KUKA KRL program: ab_com_01_st01_g01_OT.src, ab_com_01_st01_g01_OT.dat

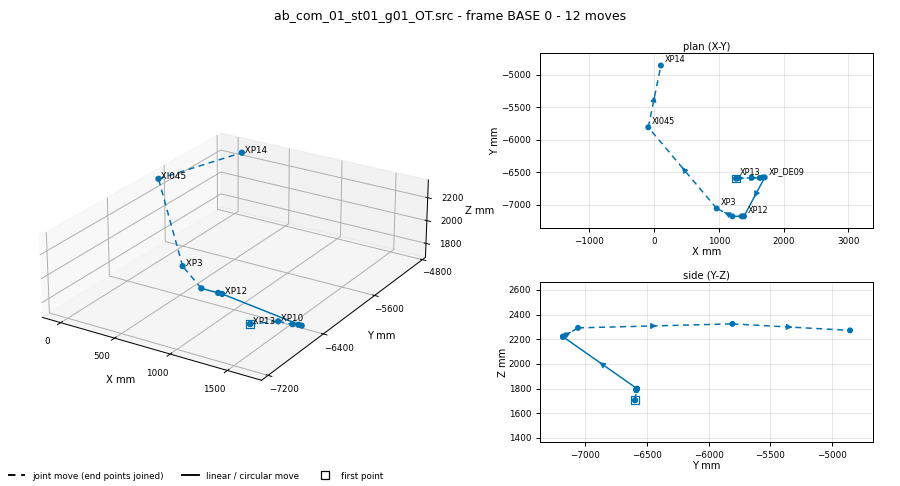
[picture p0: tool path of ab_com_01_st01_g01_OT.src in frame BASE 0, 12 of 12 moves have a stored position in this frame; points joined in program order, loops and branches not executed]
--- ab_com_01_st01_g01_OT.src ---
&ACCESS RVO1
&REL 6
&COMMENT Dep travessa LCA
&PARAM DISKPATH = KRC:\R1\Program\olp
&PARAM TEMPLATE = C:\KRC\Roboter\Template\vorgabe
&PARAM EDITMASK = *
DEF ab_com_01_st01_g01_OT( )
;FOLD INI
  ;FOLD BASISTECH INI
    GLOBAL INTERRUPT DECL 3 WHEN $STOPMESS==TRUE DO IR_STOPM ( )
    INTERRUPT ON 3
    BAS (#INITMOV,0)
  ;ENDFOLD (BASISTECH INI)
;FOLD GRIPPERTECH INI
USER_GRP(0,DUMMY,DUMMY,GDEFAULT)
;ENDFOLD (GRIPPERTECH INI)
  ;FOLD USER INI
    ;Make your modifications here

  ;ENDFOLD (USER INI)
;ENDFOLD (INI)

; Caracterizacao dos meios de producao
; Changes: Deposita LCA na GeoBox
; Modelos: Axor/Atego - ETB/LTA/LTB/STB
; Versao Atual: 30/03/2016
; Name: P13.050-R3

chk_w6_wechs_ok ( )     ; CHECK GRIPPER AXOR/ATEGO

;FOLD PTP P13 CONT Vel=100 % PDAT11 Tool[8]:Tool Changer Base[0];%{PE}%R 8.2.20,%MKUKATPBASIS,%CMOVE,%VPTP,%P 1:PTP, 2:P13, 3:C_DIS, 5:100, 7:PDAT11
$BWDSTART=FALSE
PDAT_ACT=PPDAT11
FDAT_ACT=FP13
BAS(#PTP_PARAMS,100)
PTP XP13 C_DIS
;ENDFOLD

; ABRE GRAMPOS e VERIFICA
;FOLD SET Z2.1 RPS AXOR State=OPN CONT at START Delay=1 ms;%{PE}%R 8.2.1,%MKUKATPGRP,%CGRP,%VGRP,%P 2:10, 4:1, 5:#YES, 6:GDAT26, 8:0, 10:1
TRIGGER WHEN DISTANCE=0 DELAY=1 DO H50(GRP_APO,10,1,GCONT) PRIO=-1
;ENDFOLD
;FOLD SET Z3.1 GRP AXOR State=OPN CONT at START Delay=1 ms;%{PE}%R 8.2.1,%MKUKATPGRP,%CGRP,%VGRP,%P 2:11, 4:1, 5:#YES, 6:GDAT27, 8:0, 10:1
TRIGGER WHEN DISTANCE=0 DELAY=1 DO H50(GRP_APO,11,1,GCONT) PRIO=-1
;ENDFOLD
;FOLD SET Z5.1/2/3/4 GRP AXOR State=OPN CONT at START Delay=1 ms;%{PE}%R 8.2.1,%MKUKATPGRP,%CGRP,%VGRP,%P 2:13, 4:1, 5:#YES, 6:GDAT28, 8:0, 10:1
TRIGGER WHEN DISTANCE=0 DELAY=1 DO H50(GRP_APO,13,1,GCONT) PRIO=-1
;ENDFOLD
;FOLD SET Z6.1/2/3/4 GRP AXOR State=OPN CONT at START Delay=1 ms;%{PE}%R 8.2.1,%MKUKATPGRP,%CGRP,%VGRP,%P 2:14, 4:1, 5:#YES, 6:GDAT29, 8:0, 10:1
TRIGGER WHEN DISTANCE=0 DELAY=1 DO H50(GRP_APO,14,1,GCONT) PRIO=-1
;ENDFOLD
;FOLD SET Z7.1/2 GRP AXOR State=OPN CONT at START Delay=1 ms;%{PE}%R 8.2.1,%MKUKATPGRP,%CGRP,%VGRP,%P 2:15, 4:1, 5:#YES, 6:GDAT30, 8:0, 10:1
TRIGGER WHEN DISTANCE=0 DELAY=1 DO H50(GRP_APO,15,1,GCONT) PRIO=-1
;ENDFOLD
chk_w6_rps2_opn()
chk_w6_grp3_opn()
chk_w6_grp5_opn()
chk_w6_grp6_opn()
chk_w6_grp7_opn()

;FOLD OUT 3374 'Lib. Dep. Axor/Atego' State=TRUE ;%{PE}%R 8.2.20,%MKUKATPBASIS,%COUT,%VOUTX,%P 2:3374, 3:Lib. Dep. Axor/Atego, 5:TRUE, 6:
$OUT[3374]=TRUE
;ENDFOLD
;FOLD WAIT FOR ( IN 3374 'Lib. Deposito Axor/Atego' );%{PE}%R 8.2.20,%MKUKATPBASIS,%CEXT_WAIT_FOR,%VEXT_WAIT_FOR,%P 2:, 4:, 5:$IN, 6:3374, 7:Lib. Deposito Axor/Atego, 9:
WAIT FOR  ( $IN[3374] )
;ENDFOLD
;FOLD OUT 3374 'Lib. Dep. Axor/Atego' State=FALSE ;%{PE}%R 8.2.20,%MKUKATPBASIS,%COUT,%VOUTX,%P 2:3374, 3:Lib. Dep. Axor/Atego, 5:FALSE, 6:
$OUT[3374]=FALSE
;ENDFOLD

;FOLD ; LIGA INTERLOCK 5 COM R5 com a garra rolete;%{PE}%R 8.2.20,%MKUKATPBASIS,%CCOMMENT,%VNORMAL,%P 2:LIGA  INTERLOCK  5  COM  R5  com  a  garra  rolete
;ENDFOLD
;FOLD Collision.Monitoring_5_On ;%{PE}%MKUKATPUSER
COLLSTOP( 5, 1 ) ;Interrupt-Controlled
;ENDFOLD

;FOLD PTP P9 CONT Vel=100 % PDAT7 Tool[8]:Tool Changer Base[0];%{PE}%R 8.2.20,%MKUKATPBASIS,%CMOVE,%VPTP,%P 1:PTP, 2:P9, 3:C_DIS, 5:100, 7:PDAT7
$BWDSTART=FALSE
PDAT_ACT=PPDAT7
FDAT_ACT=FP9
BAS(#PTP_PARAMS,100)
PTP XP9 C_DIS
;ENDFOLD
;FOLD PTP P10 CONT Vel=100 % PDAT8 Tool[8]:Tool Changer Base[0];%{PE}%R 8.2.20,%MKUKATPBASIS,%CMOVE,%VPTP,%P 1:PTP, 2:P10, 3:C_DIS, 5:100, 7:PDAT8
$BWDSTART=FALSE
PDAT_ACT=PPDAT8
FDAT_ACT=FP10
BAS(#PTP_PARAMS,100)
PTP XP10 C_DIS
;ENDFOLD

; VERIFICA PRESENCA LCA OK
IF (NOT(GHOST())) THEN
;FOLD WAIT FOR ( IN 489 'Presença de peça 1 - Axor LCA' );%{PE}%R 8.2.20,%MKUKATPBASIS,%CEXT_WAIT_FOR,%VEXT_WAIT_FOR,%P 2:, 4:, 5:$IN, 6:489, 7:Presença de peça 1 - Axor LCA, 9:
WAIT FOR  ( $IN[489] )
;ENDFOLD
ENDIF

; ABRE GRAMPO Z4.1 "LCA"
;FOLD SET Z4.1 GRP AXOR State=OPN CONT at START Delay=1 ms;%{PE}%R 8.2.1,%MKUKATPGRP,%CGRP,%VGRP,%P 2:12, 4:1, 5:#YES, 6:GDAT32, 8:0, 10:1
TRIGGER WHEN DISTANCE=0 DELAY=1 DO H50(GRP_APO,12,1,GCONT) PRIO=-1
;ENDFOLD

;FOLD PTP l035 CONT Vel=100 % P_OLP8 Tool[8]:Tool Changer Base[0];%{PE}%R 8.2.20,%MKUKATPBASIS,%CMOVE,%VPTP,%P 1:PTP, 2:l035, 3:C_DIS, 5:100, 7:P_OLP8
$BWDSTART=FALSE
PDAT_ACT=PP_OLP8
FDAT_ACT=Fl035
BAS(#PTP_PARAMS,100)
PTP Xl035 C_DIS
;ENDFOLD
;FOLD LIN P1 CONT Vel=0.5 m/s CPDAT1 Tool[8]:Tool Changer Base[0];%{PE}%R 8.2.20,%MKUKATPBASIS,%CMOVE,%VLIN,%P 1:LIN, 2:P1, 3:C_DIS C_DIS, 5:0.5, 7:CPDAT1
$BWDSTART=FALSE
LDAT_ACT=LCPDAT1
FDAT_ACT=FP1
BAS(#CP_PARAMS,0.5)
LIN XP1 C_DIS C_DIS
;ENDFOLD

; VERIFICA GRAMPO Z4.1 ABERTO
chk_w6_grp4_opn( )

;FOLD ; Posicao de deposito Gripper AXOR;%{PE}%R 8.2.20,%MKUKATPBASIS,%CCOMMENT,%VNORMAL,%P 2:Posicao de deposito Gripper AXOR
;ENDFOLD
;FOLD LIN P_DE09  Vel=0.25 m/s L_OLP1 Tool[6]:Gripper AXOR Base[0];%{PE}%R8.2.19,%MKUKATPBASIS,%CMOVE,%VLIN,%P 1:LIN, 2:P_DE09, 3: , 5:0.25, 7:L_OLP1
$BWDSTART = FALSE
LDAT_ACT= LL_OLP1
FDAT_ACT= FP_DE09
BAS(#CP_PARAMS,0.25)
LIN XP_DE09
;ENDFOLD

IF (NOT(GHOST())) THEN
;FOLD WAIT FOR ( IN 490 'Presença de peça 2 - Axor' AND IN 491 'Presença de peça 3 - Axor' AND IN 492 'Presença de peça 4 - Axor' );%{PE}%R 8.2.20,%MKUKATPBASIS,%CEXT_WAIT_FOR,%VEXT_WAIT_FOR,%P 2:, 4:, 5:$IN, 6:490, 7:Presença de peça 2 - Axor, 8:AND, 9:, 10:$IN, 11:491, 12:Presença de peça 3 - Axor, 13:AND, 14:, 15:$IN, 16:492, 17:Presença de peça 4 - Axor, 19:
WAIT FOR  ( $IN[490] AND $IN[491] AND $IN[492] )
;ENDFOLD
ENDIF

;FOLD OUT 3375 'Lib. p/ sair s/ Gripper Axor/Atego' State=TRUE ;%{PE}%R 8.2.20,%MKUKATPBASIS,%COUT,%VOUTX,%P 2:3375, 3:Lib. p/ sair s/ Gripper Axor/Atego, 5:TRUE, 6:
$OUT[3375]=TRUE
;ENDFOLD

; VERIFICA PRESENCA LCA OK
IF (NOT(GHOST())) THEN
;FOLD WAIT FOR ( IN 489 'Presença de peça 1 - Axor LCA' );%{PE}%R 8.2.20,%MKUKATPBASIS,%CEXT_WAIT_FOR,%VEXT_WAIT_FOR,%P 2:, 4:, 5:$IN, 6:489, 7:Presença de peça 1 - Axor LCA, 9:
WAIT FOR  ( $IN[489] )
;ENDFOLD
ENDIF

; FECHA GRAMPOS
;FOLD SET Z2.1 RPS AXOR State=CLO GDAT15;%{PE}%R 8.2.1,%MKUKATPGRP,%CGRP,%VGRP,%P 2:10, 4:2, 5:#NO, 6:GDAT15, 8:0, 10:0
H50(GRP,10,2,GGDAT15)
;ENDFOLD
;FOLD SET Z3.1 GRP AXOR State=CLO GDAT8;%{PE}%R 8.2.1,%MKUKATPGRP,%CGRP,%VGRP,%P 2:11, 4:2, 5:#NO, 6:GDAT8, 8:0, 10:0
H50(GRP,11,2,GGDAT8)
;ENDFOLD
;FOLD SET Z5.1/2/3/4 GRP AXOR State=CLO GDAT16;%{PE}%R 8.2.1,%MKUKATPGRP,%CGRP,%VGRP,%P 2:13, 4:2, 5:#NO, 6:GDAT16, 8:0, 10:0
H50(GRP,13,2,GGDAT16)
;ENDFOLD
;FOLD SET Z6.1/2/3/4 GRP AXOR State=CLO GDAT17;%{PE}%R 8.2.1,%MKUKATPGRP,%CGRP,%VGRP,%P 2:14, 4:2, 5:#NO, 6:GDAT17, 8:0, 10:0
H50(GRP,14,2,GGDAT17)
;ENDFOLD

; VERIFICA GRAMPOS FECHADOS
chk_w6_rps2_clo( )
chk_w6_grp3_clo( )

; FECHA GRAMPOS Z4.1 e Z7.1
;FOLD SET Z4.1 GRP AXOR State=CLO GDAT31;%{PE}%R 8.2.1,%MKUKATPGRP,%CGRP,%VGRP,%P 2:12, 4:2, 5:#NO, 6:GDAT31, 8:0, 10:0
H50(GRP,12,2,GGDAT31)
;ENDFOLD
;FOLD SET Z7.1/2 GRP AXOR State=CLO GDAT33;%{PE}%R 8.2.1,%MKUKATPGRP,%CGRP,%VGRP,%P 2:15, 4:2, 5:#NO, 6:GDAT33, 8:0, 10:0
H50(GRP,15,2,GGDAT33)
;ENDFOLD
;FOLD SET VACUO AXOR State=BLOW GDAT34;%{PE}%R 8.2.1,%MKUKATPGRP,%CGRP,%VGRP,%P 2:9, 4:2, 5:#NO, 6:GDAT34, 8:0, 10:0
H50(GRP,9,2,GGDAT34)
;ENDFOLD
;FOLD SET VACUO AXOR State=OFF GDAT35;%{PE}%R 8.2.1,%MKUKATPGRP,%CGRP,%VGRP,%P 2:9, 4:3, 5:#NO, 6:GDAT35, 8:0, 10:0
H50(GRP,9,3,GGDAT35)
;ENDFOLD

; VERIFICA GRAMPOS FECHADOS
chk_w6_grp5_clo( )
chk_w6_grp6_clo( )
chk_w6_grp7_clo( )
chk_w6_grp4_clo( )
chk_w6_grp1_vacoff( )

; VERIFICA PRESENCA LCA OK
IF (NOT(GHOST())) THEN
;FOLD WAIT FOR ( IN 489 'Presença de peça 1 - Axor LCA' );%{PE}%R 8.2.20,%MKUKATPBASIS,%CEXT_WAIT_FOR,%VEXT_WAIT_FOR,%P 2:, 4:, 5:$IN, 6:489, 7:Presença de peça 1 - Axor LCA, 9:
WAIT FOR  ( $IN[489] )
;ENDFOLD
ENDIF

;FOLD OUT 3375 'Lib. p/ sair s/ Gripper Axor/Atego' State=TRUE ;%{PE}%R 8.2.20,%MKUKATPBASIS,%COUT,%VOUTX,%P 2:3375, 3:Lib. p/ sair s/ Gripper Axor/Atego, 5:TRUE, 6:
$OUT[3375]=TRUE
;ENDFOLD
;FOLD WAIT FOR ( IN 3375 'Lib. p/ sair s/ Gripper Axor/Atego' );%{PE}%R 8.2.20,%MKUKATPBASIS,%CEXT_WAIT_FOR,%VEXT_WAIT_FOR,%P 2:, 4:, 5:$IN, 6:3375, 7:Lib. p/ sair s/ Gripper Axor/Atego, 9:
WAIT FOR  ( $IN[3375] )
;ENDFOLD
;FOLD OUT 3375 'Lib. p/ sair s/ Gripper Axor/Atego' State=FALSE ;%{PE}%R 8.2.20,%MKUKATPBASIS,%COUT,%VOUTX,%P 2:3375, 3:Lib. p/ sair s/ Gripper Axor/Atego, 5:FALSE, 6:
$OUT[3375]=FALSE
;ENDFOLD

;FOLD WAIT Time=0.5 sec;%{PE}%R 8.2.20,%MKUKATPBASIS,%CWAIT,%VWAIT,%P 3:0.5
WAIT SEC 0.5
;ENDFOLD
;FOLD OUT 224 'Bloquear MPS' State=FALSE ;%{PE}%R 8.2.20,%MKUKATPBASIS,%COUT,%VOUTX,%P 2:224, 3:Bloquear MPS, 5:FALSE, 6:
$OUT[224]=FALSE
;ENDFOLD
;FOLD OUT 223 'Desbloquear MPS' State=TRUE ;%{PE}%R 8.2.20,%MKUKATPBASIS,%COUT,%VOUTX,%P 2:223, 3:Desbloquear MPS, 5:TRUE, 6:
$OUT[223]=TRUE
;ENDFOLD
;FOLD WAIT FOR ( IN 217 'MPS Destravado' );%{PE}%R 8.2.20,%MKUKATPBASIS,%CEXT_WAIT_FOR,%VEXT_WAIT_FOR,%P 2:, 4:, 5:$IN, 6:217, 7:MPS Destravado, 9:
WAIT FOR  ( $IN[217] )
;ENDFOLD
;FOLD WAIT FOR NOT ( IN 221 'MPS Travado' );%{PE}%R 8.2.20,%MKUKATPBASIS,%CEXT_WAIT_FOR,%VEXT_WAIT_FOR,%P 2:NOT, 4:, 5:$IN, 6:221, 7:MPS Travado, 9:
WAIT FOR  NOT ( $IN[221] )
;ENDFOLD
;FOLD IBUS OFF;%{PE}%R 8.2.20,%MKUKATPBASIS,%CIBUS,%VMAP,%P 2:#OFF, 3:3
$IBUS_OFF=$IBUS_ON
$IBUS_ON=0
;ENDFOLD
;FOLD WAIT Time=0.5 sec;%{PE}%R 8.2.20,%MKUKATPBASIS,%CWAIT,%VWAIT,%P 3:0.5
WAIT SEC 0.5
;ENDFOLD

;FOLD LIN P12 Vel=0.25 m/s CPDAT6 Tool[8]:Tool Changer Base[0];%{PE}%R 8.2.20,%MKUKATPBASIS,%CMOVE,%VLIN,%P 1:LIN, 2:P12, 3:, 5:0.25, 7:CPDAT6
$BWDSTART=FALSE
LDAT_ACT=LCPDAT6
FDAT_ACT=FP12
BAS(#CP_PARAMS,0.25)
LIN XP12
;ENDFOLD

;FOLD WAIT FOR NOT ( IN 219 'Posicao p/ Acoplamento OK' );%{PE}%R 8.2.20,%MKUKATPBASIS,%CEXT_WAIT_FOR,%VEXT_WAIT_FOR,%P 2:NOT, 4:, 5:$IN, 6:219, 7:Posicao p/ Acoplamento OK, 9:
WAIT FOR  NOT ( $IN[219] )
;ENDFOLD

;FOLD LIN l040 Vel=0.25 m/s L_OLP2 Tool[8]:Tool Changer Base[0];%{PE}%R 8.2.20,%MKUKATPBASIS,%CMOVE,%VLIN,%P 1:LIN, 2:l040, 3:, 5:0.25, 7:L_OLP2
$BWDSTART=FALSE
LDAT_ACT=LL_OLP2
FDAT_ACT=Fl040
BAS(#CP_PARAMS,0.25)
LIN Xl040
;ENDFOLD

;FOLD WAIT FOR NOT ( IN 219 'Posicao p/ Acoplamento OK' );%{PE}%R 8.2.20,%MKUKATPBASIS,%CEXT_WAIT_FOR,%VEXT_WAIT_FOR,%P 2:NOT, 4:, 5:$IN, 6:219, 7:Posicao p/ Acoplamento OK, 9:
WAIT FOR  NOT ( $IN[219] )
;ENDFOLD
;FOLD OUT 223 'Desbloquear MPS' State=FALSE ;%{PE}%R 8.2.20,%MKUKATPBASIS,%COUT,%VOUTX,%P 2:223, 3:Desbloquear MPS, 5:FALSE, 6:
$OUT[223]=FALSE
;ENDFOLD

;FOLD LIN P2 CONT Vel=1 m/s CPDAT2 Tool[8]:Tool Changer Base[0];%{PE}%R 8.2.20,%MKUKATPBASIS,%CMOVE,%VLIN,%P 1:LIN, 2:P2, 3:C_DIS C_DIS, 5:1, 7:CPDAT2
$BWDSTART=FALSE
LDAT_ACT=LCPDAT2
FDAT_ACT=FP2
BAS(#CP_PARAMS,1)
LIN XP2 C_DIS C_DIS
;ENDFOLD
;FOLD PTP P3 CONT Vel=100 % PDAT1 Tool[8]:Tool Changer Base[0];%{PE}%R 8.2.20,%MKUKATPBASIS,%CMOVE,%VPTP,%P 1:PTP, 2:P3, 3:C_DIS, 5:100, 7:PDAT1
$BWDSTART=FALSE
PDAT_ACT=PPDAT1
FDAT_ACT=FP3
BAS(#PTP_PARAMS,100)
PTP XP3 C_DIS
;ENDFOLD
;FOLD PTP l045 CONT Vel=100 % P_OLP9 Tool[8]:Tool Changer Base[0];%{PE}%R 8.2.20,%MKUKATPBASIS,%CMOVE,%VPTP,%P 1:PTP, 2:l045, 3:C_DIS, 5:100, 7:P_OLP9
$BWDSTART=FALSE
PDAT_ACT=PP_OLP9
FDAT_ACT=Fl045
BAS(#PTP_PARAMS,100)
PTP Xl045 C_DIS
;ENDFOLD

;FOLD PULSE 3343 'R3 entregou peça Geo' State=TRUE Time=3 sec;%{PE}%R 8.2.20,%MKUKATPBASIS,%COUT,%VPULSE,%P 2:3343, 3:R3 entregou peça Geo, 5:TRUE, 6:, 8:3
PULSE($OUT[3343], TRUE,3)
;ENDFOLD

;FOLD PTP P14 CONT Vel=100 % PDAT12 Tool[8]:Tool Changer Base[0];%{PE}%R 8.2.20,%MKUKATPBASIS,%CMOVE,%VPTP,%P 1:PTP, 2:P14, 3:C_DIS, 5:100, 7:PDAT12
$BWDSTART=FALSE
PDAT_ACT=PPDAT12
FDAT_ACT=FP14
BAS(#PTP_PARAMS,100)
PTP XP14 C_DIS
;ENDFOLD

;FOLD ; DESLIGA INTERLOCK 1 COM R1 NA PEGA DA GARRA 913;%{PE}%R 8.2.20,%MKUKATPBASIS,%CCOMMENT,%VNORMAL,%P 2:DESLIGA  INTERLOCK  1  COM  R1  NA  PEGA  DA  GARRA  913
;ENDFOLD
;FOLD Collision.Monitoring_1_Off . ;%{PE}%MKUKATPUSER
COLLSTOP( 1, 2+0 )
;ENDFOLD

;FOLD ; DESLIGA INTERLOCK 5 COM R5;%{PE}%R 8.2.20,%MKUKATPBASIS,%CCOMMENT,%VNORMAL,%P 2:DESLIGA  INTERLOCK  5  COM  R5
;ENDFOLD
;FOLD Collision.Monitoring_5_Off . ;%{PE}%MKUKATPUSER
COLLSTOP( 5, 2+0 )
;ENDFOLD

;FOLD OUT 3374 'Lib. Dep. Axor/Atego' State=TRUE ;%{PE}%R 8.2.20,%MKUKATPBASIS,%COUT,%VOUTX,%P 2:3374, 3:Lib. Dep. Axor/Atego, 5:TRUE, 6:
$OUT[3374]=TRUE
;ENDFOLD
;FOLD OUT 3348 'Fora area GEOBOX' State=TRUE ;%{PE}%R 8.2.20,%MKUKATPBASIS,%COUT,%VOUTX,%P 2:3348, 3:Fora area GEOBOX, 5:TRUE, 6:
$OUT[3348]=TRUE
;ENDFOLD

END

--- ab_com_01_st01_g01_OT.dat ---
&ACCESS RVO1
&REL 6
&COMMENT Dep travessa LCA
&PARAM DISKPATH = KRC:\R1\Program\olp
&PARAM TEMPLATE = C:\KRC\Roboter\Template\vorgabe
&PARAM EDITMASK = *
DEFDAT  ab_com_01_st01_g01_OT
;FOLD EXTERNAL DECLARATIONS;%{PE}%MKUKATPBASIS,%CEXT,%VCOMMON,%P
;FOLD GRIPPERTECH EXT
EXT  H50 (INT  :IN,INT  :IN,INT  :IN,GRP_TYP  :IN )
;ENDFOLD (GRIPPERTECH EXT)
;FOLD SPOTTECH EXT

;ENDFOLD (SPOTTECH EXT)
;FOLD BASISTECH EXT;%{PE}%MKUKATPBASIS,%CEXT,%VEXT,%P
EXT  BAS (BAS_COMMAND  :IN,REAL  :IN )
DECL INT SUCCESS
;ENDFOLD (BASISTECH EXT)
;FOLD USER EXT;%{E}%MKUKATPUSER,%CEXT,%VEXT,%P
;Make your modifications here

;ENDFOLD (USER EXT)
;ENDFOLD (EXTERNAL DECLARATIONS)
DECL FDAT Fl035={TOOL_NO 6,BASE_NO 0,IPO_FRAME #BASE,POINT2[] " "}
DECL PDAT PP_OLP8={VEL 100.0,ACC 100.0,APO_DIST 100.0,APO_MODE #CDIS}
DECL E6POS Xl035={X 1631.40002,Y -6588.3291,Z 1794.03101,A 70.7797089,B -89.9868469,C -175.781799,S 6,T 51,E1 5700.0,E2 0.0,E3 0.0,E4 0.0,E5 0.0,E6 0.0}
DECL FDAT FP_DE09={TOOL_NO 6,BASE_NO 0,IPO_FRAME #BASE,POINT2[] " "}
DECL E6POS XP_DE09={X 1707.35596,Y -6580.3291,Z 1798.76196,A -108.196297,B -89.8673096,C 3.225034,S 6,T 51,E1 5699.99805,E2 0.0,E3 0.0,E4 0.0,E5 0.0,E6 0.0}
DECL LDAT LL_OLP1={VEL 0.25,ACC 100.0,APO_DIST 0.0,APO_FAC 0.0,ORI_TYP #VAR,CIRC_TYP #BASE,JERK_FAC 50.0}
DECL FDAT Fl040={TOOL_NO 8,BASE_NO 0,IPO_FRAME #BASE,POINT2[] " ",TQ_STATE FALSE}
DECL E6POS Xl040={X 1353.49902,Y -7181.71094,Z 2220.25488,A -90.1084976,B -74.8772964,C -89.8598785,S 6,T 51,E1 5700.01904,E2 0.0,E3 0.0,E4 0.0,E5 0.0,E6 0.0}
DECL LDAT LL_OLP2={VEL 0.25,ACC 100.0,APO_DIST 20.0,APO_FAC 0.0,ORI_TYP #VAR,CIRC_TYP #BASE,JERK_FAC 50.0}
DECL FDAT Fl045={TOOL_NO 8,BASE_NO 0,IPO_FRAME #BASE,POINT2[] " "}
DECL PDAT PP_OLP9={VEL 100.0,ACC 100.0,APO_DIST 100.0,APO_MODE #CDIS}
DECL E6POS Xl045={X -89.0451508,Y -5808.14014,Z 2324.49902,A 10.4492998,B 8.6899004,C 149.959503,S 6,T 51,E1 4593.48291,E2 0.0,E3 0.0,E4 0.0,E5 0.0,E6 0.0}
DECL BASIS_SUGG_T LAST_BASIS={POINT1[] "P0                      ",POINT2[] "P0                      ",CP_PARAMS[] "CPDAT0                  ",PTP_PARAMS[] "PDAT0                   ",CONT[] "                        ",CP_VEL[] "2.0                     ",PTP_VEL[] " 100                    ",SYNC_PARAMS[] "SYNCDAT                 ",SPL_NAME[] "S0                      "}
DECL E6POS XP1={X 1678.87805,Y -6580.3291,Z 1798.76196,A -108.197998,B -89.8673096,C 3.226717,S 6,T 51,E1 5699.99805,E2 0.0,E3 0.0,E4 0.0,E5 0.0,E6 0.0}
DECL FDAT FP1={TOOL_NO 6,BASE_NO 0,IPO_FRAME #BASE,POINT2[] " ",TQ_STATE FALSE}
DECL LDAT LCPDAT1={VEL 2.0,ACC 100.0,APO_DIST 50.0,APO_FAC 50.0,AXIS_VEL 100.0,AXIS_ACC 100.0,ORI_TYP #VAR,CIRC_TYP #BASE,JERK_FAC 50.0,GEAR_JERK 50.0,EXAX_IGN 0}
DECL E6POS XP2={X 1208.60706,Y -7181.56104,Z 2220.479,A -89.9195328,B -74.9438934,C -90.0642395,S 6,T 51,E1 5699.41699,E2 0.0,E3 0.0,E4 0.0,E5 0.0,E6 0.0}
DECL FDAT FP2={TOOL_NO 8,BASE_NO 0,IPO_FRAME #BASE,POINT2[] " ",TQ_STATE FALSE}
DECL LDAT LCPDAT2={VEL 2.0,ACC 100.0,APO_DIST 100.0,APO_FAC 50.0,AXIS_VEL 100.0,AXIS_ACC 100.0,ORI_TYP #VAR,CIRC_TYP #BASE,JERK_FAC 50.0,GEAR_JERK 50.0,EXAX_IGN 0}
DECL E6POS XP3={X 965.776001,Y -7059.44189,Z 2292.1189,A -54.9305382,B -71.0292969,C -129.947205,S 6,T 51,E1 5619.95313,E2 0.0,E3 0.0,E4 0.0,E5 0.0,E6 0.0}
DECL FDAT FP3={TOOL_NO 8,BASE_NO 0,IPO_FRAME #BASE,POINT2[] " ",TQ_STATE FALSE}
DECL PDAT PPDAT1={VEL 100.0,ACC 100.0,APO_DIST 100.0,APO_MODE #CDIS}
DECL GRP_SUGG_T LAST_GRP={NUMBER[] "9                       ",STATE[] "3                       ",PARAMS[] "GDAT35                  "}
DECL GRP_TYP GGDAT2={G_APO #NO,GRP_TIME 0.200000003,CTRL #OFF,DLY 0,DST 1}
DECL GRP_TYP GGDAT1={G_APO #NO,GRP_TIME 0.200000003,CTRL #OFF,DLY 0,DST 1}
DECL GRP_TYP GGDAT3={G_APO #NO,GRP_TIME 0.200000003,CTRL #OFF,DLY 0,DST 1}
DECL GRP_TYP GGDAT4={G_APO #NO,GRP_TIME 0.200000003,CTRL #OFF,DLY 0,DST 1}
DECL GRP_TYP GGDAT5={G_APO #NO,GRP_TIME 0.200000003,CTRL #OFF,DLY 0,DST 1}
DECL GRP_TYP GGDAT6={G_APO #NO,GRP_TIME 0.200000003,CTRL #OFF,DLY 0,DST 1}
DECL GRP_TYP GGDAT7={G_APO #NO,GRP_TIME 0.200000003,CTRL #OFF,DLY 0,DST 1}
DECL GRP_TYP GGDAT8={G_APO #NO,GRP_TIME 0.200000003,CTRL #OFF,DLY 0,DST 1}
DECL GRP_TYP GGDAT9={G_APO #NO,GRP_TIME 0.200000003,CTRL #OFF,DLY 0,DST 1}
DECL GRP_TYP GGDAT10={G_APO #NO,GRP_TIME 0.200000003,CTRL #OFF,DLY 0,DST 1}
DECL GRP_TYP GGDAT11={G_APO #NO,GRP_TIME 0.200000003,CTRL #OFF,DLY 0,DST 1}
DECL GRP_TYP GGDAT12={G_APO #NO,GRP_TIME 0.200000003,CTRL #OFF,DLY 0,DST 1}
DECL GRP_TYP GGDAT13={G_APO #NO,GRP_TIME 0.200000003,CTRL #OFF,DLY 0,DST 1}
DECL GRP_TYP GGDAT14={G_APO #NO,GRP_TIME 0.200000003,CTRL #OFF,DLY 0,DST 1}
DECL GRP_TYP GGDAT15={G_APO #NO,GRP_TIME 0.200000003,CTRL #OFF,DLY 0,DST 1}
DECL GRP_TYP GGDAT16={G_APO #NO,GRP_TIME 0.200000003,CTRL #OFF,DLY 0,DST 1}
DECL GRP_TYP GGDAT17={G_APO #NO,GRP_TIME 0.200000003,CTRL #OFF,DLY 0,DST 1}
DECL GRP_TYP GGDAT18={G_APO #NO,GRP_TIME 0.200000003,CTRL #OFF,DLY 0,DST 1}
DECL GRP_TYP GGDAT19={G_APO #NO,GRP_TIME 0.200000003,CTRL #OFF,DLY 0,DST 1}
DECL E6POS XP8={X 846.208923,Y -6811.92188,Z 1735.02002,A -9.90643406,B -75.1019363,C -110.246101,S 6,T 51,E1 5398.51416,E2 0.0,E3 0.0,E4 0.0,E5 0.0,E6 0.0}
DECL FDAT FP8={TOOL_NO 6,BASE_NO 0,IPO_FRAME #BASE,POINT2[] " ",TQ_STATE FALSE}
DECL PDAT PPDAT6={VEL 100.0,ACC 100.0,APO_DIST 100.0,APO_MODE #CDIS}
DECL E6POS XP9={X 1266.59302,Y -6597.0752,Z 1705.35596,A 1.41324604,B -82.7240829,C -106.323402,S 6,T 51,E1 5699.94922,E2 0.0,E3 0.0,E4 0.0,E5 0.0,E6 0.0}
DECL FDAT FP9={TOOL_NO 6,BASE_NO 0,IPO_FRAME #BASE,POINT2[] " ",TQ_STATE FALSE}
DECL PDAT PPDAT7={VEL 100.0,ACC 100.0,APO_DIST 100.0,APO_MODE #CDIS}
DECL E6POS XP10={X 1506.66797,Y -6587.14014,Z 1785.50403,A 0.0,B -89.9998932,C -105.000099,S 6,T 51,E1 5700.0,E2 0.0,E3 0.0,E4 0.0,E5 0.0,E6 0.0}
DECL FDAT FP10={TOOL_NO 6,BASE_NO 0,IPO_FRAME #BASE,POINT2[] " ",TQ_STATE FALSE}
DECL PDAT PPDAT8={VEL 100.0,ACC 100.0,APO_DIST 100.0,APO_MODE #CDIS}
DECL GRP_TYP GGDAT20={G_APO #NO,GRP_TIME 0.200000003,CTRL #OFF,DLY 0,DST 1}
DECL GRP_TYP GGDAT21={G_APO #NO,GRP_TIME 0.200000003,CTRL #OFF,DLY 0,DST 1}
DECL GRP_TYP GGDAT22={G_APO #NO,GRP_TIME 0.200000003,CTRL #OFF,DLY 0,DST 1}
DECL GRP_TYP GGDAT23={G_APO #NO,GRP_TIME 0.200000003,CTRL #OFF,DLY 0,DST 1}
DECL GRP_TYP GGDAT24={G_APO #NO,GRP_TIME 0.200000003,CTRL #OFF,DLY 0,DST 1}
DECL GRP_TYP GGDAT25={G_APO #NO,GRP_TIME 0.200000003,CTRL #OFF,DLY 0,DST 1}
DECL GRP_TYP GGDAT26={G_APO #NO,GRP_TIME 0.200000003,CTRL #OFF,DLY 0,DST 1}
DECL GRP_TYP GGDAT27={G_APO #NO,GRP_TIME 0.200000003,CTRL #OFF,DLY 0,DST 1}
DECL GRP_TYP GGDAT28={G_APO #NO,GRP_TIME 0.200000003,CTRL #OFF,DLY 0,DST 1}
DECL GRP_TYP GGDAT29={G_APO #NO,GRP_TIME 0.200000003,CTRL #OFF,DLY 0,DST 1}
DECL GRP_TYP GGDAT30={G_APO #NO,GRP_TIME 0.200000003,CTRL #OFF,DLY 0,DST 1}
DECL E6POS XP12={X 1387.84399,Y -7181.62695,Z 2220.25806,A -90.1207123,B -74.8770218,C -89.8428421,S 6,T 51,E1 5699.97217,E2 0.0,E3 0.0,E4 0.0,E5 0.0,E6 0.0}
DECL FDAT FP12={TOOL_NO 8,BASE_NO 0,IPO_FRAME #BASE,POINT2[] " ",TQ_STATE FALSE}
DECL LDAT LCPDAT6={VEL 2.0,ACC 100.0,APO_DIST 100.0,APO_FAC 50.0,AXIS_VEL 100.0,AXIS_ACC 100.0,ORI_TYP #VAR,CIRC_TYP #BASE,JERK_FAC 50.0,GEAR_JERK 50.0,EXAX_IGN 0}
DECL E6POS XP13={X 1266.59302,Y -6597.0752,Z 1705.35596,A 1.41324604,B -82.7240829,C -106.323402,S 6,T 51,E1 5699.94922,E2 0.0,E3 0.0,E4 0.0,E5 0.0,E6 0.0}
DECL FDAT FP13={TOOL_NO 6,BASE_NO 0,IPO_FRAME #BASE,POINT2[] " ",TQ_STATE FALSE}
DECL PDAT PPDAT11={VEL 100.0,ACC 100.0,APO_DIST 100.0,APO_MODE #CDIS}
DECL E6POS XP14={X 105.763496,Y -4854.61084,Z 2271.72412,A 91.3470612,B 9.42022896,C -178.990005,S 2,T 35,E1 3441.56201,E2 0.0,E3 0.0,E4 0.0,E5 0.0,E6 0.0}
DECL FDAT FP14={TOOL_NO 8,BASE_NO 0,IPO_FRAME #BASE,POINT2[] " ",TQ_STATE FALSE}
DECL PDAT PPDAT12={VEL 100.0,ACC 100.0,APO_DIST 100.0,APO_MODE #CDIS}
DECL GRP_TYP GGDAT31={G_APO #NO,GRP_TIME 0.200000003,CTRL #OFF,DLY 0,DST 1}
DECL GRP_TYP GCONT={G_APO #YES,GRP_TIME 0.0,CTRL #OFF,DLY 0,DST 0}
DECL GRP_TYP GGDAT32={G_APO #NO,GRP_TIME 0.200000003,CTRL #OFF,DLY 0,DST 1}
DECL GRP_TYP GGDAT33={G_APO #NO,GRP_TIME 0.200000003,CTRL #OFF,DLY 0,DST 1}
DECL GRP_TYP GGDAT34={G_APO #NO,GRP_TIME 0.200000003,CTRL #OFF,DLY 0,DST 1}
DECL GRP_TYP GGDAT35={G_APO #NO,GRP_TIME 0.200000003,CTRL #OFF,DLY 0,DST 1}
ENDDAT
